FUNCTION POU_MoveToPosFunc : INT
VAR_INPUT
	actualPos : INT ;
	requiredPos : INT;
	speed: INT;

	
END_VAR
VAR
	timer : ton;
	newPos : int;
	startTimer: BOOL;
	calculatedTime: TIME;
	test : INT := 0;
	testbuitenif :int := 0;
END_VAR

startTimer:= TRUE;
calculatedTime :=INT_TO_TIME(1000/speed);
timer(in:= startTimer, pt:= calculatedTime);
testbuitenif := testbuitenif + 1;
IF timer.Q OR TRUE THEN
	test := test + 1;
	startTimer:=FALSE;
	IF requiredPos < actualpos THEN
		newpos := actualPos -1;
	ELSIF requiredpos > actualpos THEN
		newpos := actualPos +1; 
	END_IF
	POU_MoveToPosFunc := newpos;
END_IF
//pou_movetopos := newpos;
//RETURN pou_movetopos;
//pou_movetopos:= actualpos + requiredpos+speed;

END_FUNCTION

(* stored: Version 1.1.0.1, ProductVersion 3.1.4024.12
   POU POU_MoveToPosFunc: Id {f1b905d7-21a7-4edb-bcb9-64fac2a8debd}, SpecialFunc None *)
